SYSTEM DASDA1 (* System Configuration *)
  (* Standard: 61499-1 *)
  (* Version 0.4, 2009-03-05, JHC, Holobloc Inc., Deleted Application. *)
  (* Version 0.3, 2003-12-05, JHC, Rockwell Automation, Renamed from NEWSYSTEM. *)
  (* Version 0.2, 2002-11-05, JHC, Rockwell Automation, Fixed missing (empty) FBD in Application. *)
  (* Version 0.1, 2002-01-17, JHC, Rockwell Automation, Minor cleanup *)
  (* Version 0.0, 2000-05-27, JHC, Rockwell Automation *)
  DEVICE HMI_LAYER : FRAME_DEVICE(BOUNDS := [0,0,200,600])
    RESOURCE HMI_up : PANEL_RESOURCE(COLS := 1, ROWS := 10)
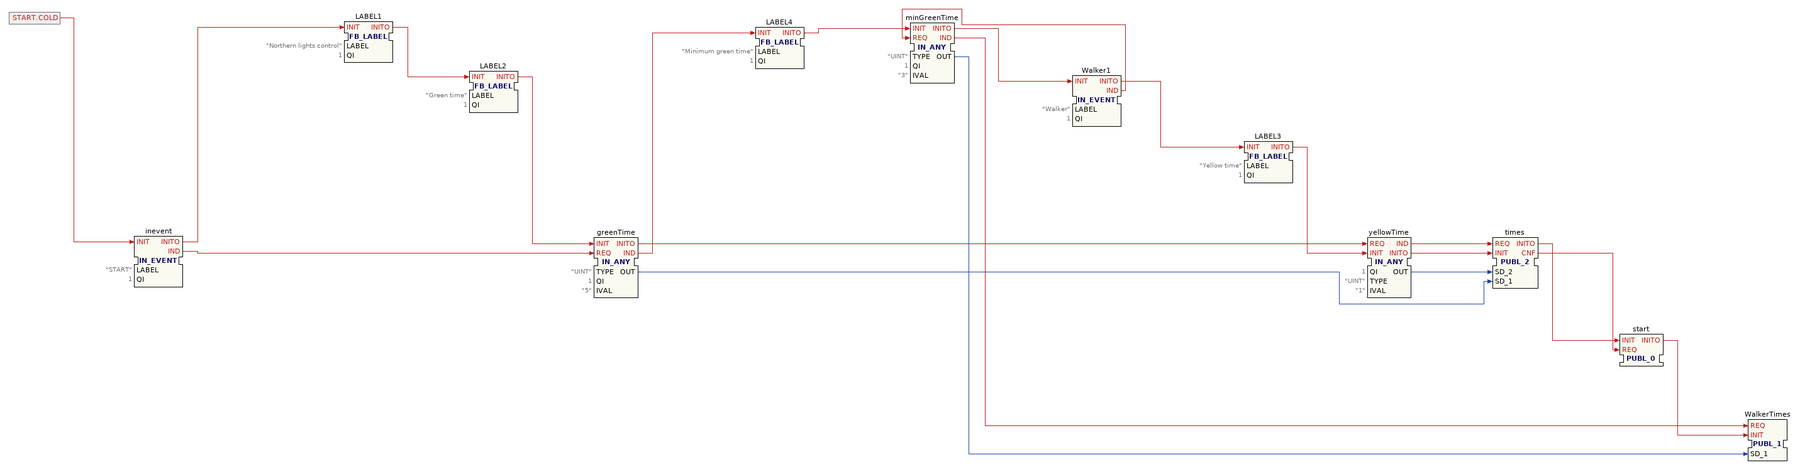
      FBS
        start : PUBL_0;
        greenTime : IN_ANY(TYPE := "UINT", QI := 1, IVAL := "5");
        yellowTime : IN_ANY(QI := 1, TYPE := "UINT", IVAL := "1");
        times : PUBL_2;
        LABEL1 : FB_LABEL(LABEL := "Northern lights control", QI := 1);
        LABEL2 : FB_LABEL(LABEL := "Green time", QI := 1);
        LABEL3 : FB_LABEL(LABEL := "Yellow time", QI := 1);
        minGreenTime : IN_ANY(TYPE := "UINT", QI := 1, IVAL := "3");
        LABEL4 : FB_LABEL(LABEL := "Minimum green time", QI := 1);
        Walker1 : IN_EVENT(LABEL := "Walker", QI := 1);
        WalkerTimes : PUBL_1;
        inevent : IN_EVENT(LABEL := "START", QI := 1);
      END_FBS
      EVENT_CONNECTIONS
        yellowTime.IND TO times.REQ;
        LABEL1.INITO TO LABEL2.INIT;
        LABEL2.INITO TO greenTime.INIT;
        greenTime.INITO TO LABEL4.INIT;
        LABEL4.INITO TO minGreenTime.INIT;
        greenTime.IND TO yellowTime.REQ;
        yellowTime.INITO TO times.INIT;
        times.INITO TO start.INIT;
        times.CNF TO start.REQ;
        minGreenTime.INITO TO Walker1.INIT;
        Walker1.INITO TO LABEL3.INIT;
        LABEL3.INITO TO yellowTime.INIT;
        Walker1.IND TO minGreenTime.REQ;
        minGreenTime.IND TO WalkerTimes.REQ;
        start.INITO TO WalkerTimes.INIT;
        START.COLD TO inevent.INIT;
        inevent.INITO TO LABEL1.INIT;
        inevent.IND TO greenTime.REQ;
      END_CONNECTIONS
      DATA_CONNECTIONS
        yellowTime.OUT TO times.SD_2;
        greenTime.OUT TO times.SD_1;
        minGreenTime.OUT TO WalkerTimes.SD_1;
      END_CONNECTIONS
    END_RESOURCE
    RESOURCE HMI_left : PANEL_RESOURCE(COLS := 1, ROWS := 10)
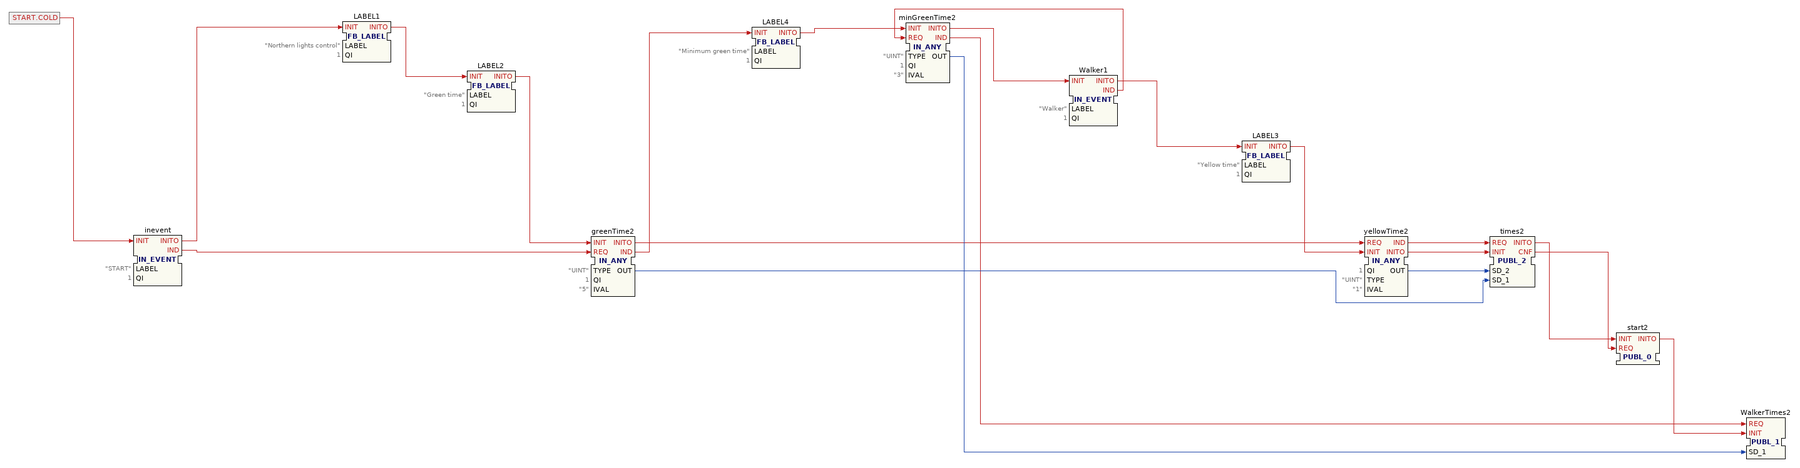
      FBS
        start2 : PUBL_0;
        greenTime2 : IN_ANY(TYPE := "UINT", QI := 1, IVAL := "5");
        yellowTime2 : IN_ANY(QI := 1, TYPE := "UINT", IVAL := "1");
        times2 : PUBL_2;
        LABEL1 : FB_LABEL(LABEL := "Northern lights control", QI := 1);
        LABEL2 : FB_LABEL(LABEL := "Green time", QI := 1);
        LABEL3 : FB_LABEL(LABEL := "Yellow time", QI := 1);
        minGreenTime2 : IN_ANY(TYPE := "UINT", QI := 1, IVAL := "3");
        LABEL4 : FB_LABEL(LABEL := "Minimum green time", QI := 1);
        Walker1 : IN_EVENT(LABEL := "Walker", QI := 1);
        WalkerTimes2 : PUBL_1;
        inevent : IN_EVENT(LABEL := "START", QI := 1);
      END_FBS
      EVENT_CONNECTIONS
        yellowTime2.IND TO times2.REQ;
        LABEL1.INITO TO LABEL2.INIT;
        LABEL2.INITO TO greenTime2.INIT;
        greenTime2.INITO TO LABEL4.INIT;
        LABEL4.INITO TO minGreenTime2.INIT;
        greenTime2.IND TO yellowTime2.REQ;
        yellowTime2.INITO TO times2.INIT;
        times2.INITO TO start2.INIT;
        times2.CNF TO start2.REQ;
        minGreenTime2.INITO TO Walker1.INIT;
        Walker1.INITO TO LABEL3.INIT;
        LABEL3.INITO TO yellowTime2.INIT;
        Walker1.IND TO minGreenTime2.REQ;
        minGreenTime2.IND TO WalkerTimes2.REQ;
        start2.INITO TO WalkerTimes2.INIT;
        START.COLD TO inevent.INIT;
        inevent.INITO TO LABEL1.INIT;
        inevent.IND TO greenTime2.REQ;
      END_CONNECTIONS
      DATA_CONNECTIONS
        yellowTime2.OUT TO times2.SD_2;
        greenTime2.OUT TO times2.SD_1;
        minGreenTime2.OUT TO WalkerTimes2.SD_1;
      END_CONNECTIONS
    END_RESOURCE
  END_DEVICE
  DEVICE MODEL_LAYER : FRAME_DEVICE
    RESOURCE LIGHTS_U : PANEL_RESOURCE
      FBS
        LightsControl : PUBL_3;
        start : SUBL_0;
        times : SUBL_2;
        LightsRT : PUBL_2;
        WalkerTimes : SUBL_1;
        LC1 : LIGHTS_CYCLE;
      END_FBS
      EVENT_CONNECTIONS
        START.COLD TO times.INIT;
        LightsControl.CNF TO LightsRT.REQ;
        start.INITO TO LightsControl.INIT;
        LightsControl.INITO TO LightsRT.INIT;
        times.INITO TO WalkerTimes.INIT;
        WalkerTimes.INITO TO start.INIT;
        start.IND TO LC1.START;
        WalkerTimes.IND TO LC1.WALKER;
        LC1.CNF TO LightsControl.REQ;
      END_CONNECTIONS
      DATA_CONNECTIONS
        WalkerTimes.RD_1 TO LC1.WALKERT;
        times.RD_1 TO LC1.GREENT;
        times.RD_2 TO LC1.YELLOWT;
        LC1.GREENOUT TO LightsControl.SD_1;
        LC1.YELLOWOUT TO LightsControl.SD_2;
        LC1.REDOUT TO LightsControl.SD_3;
        LC1.GREENRT TO LightsRT.SD_1;
        LC1.YELLOWRT TO LightsRT.SD_2;
      END_CONNECTIONS
    END_RESOURCE
    RESOURCE LIGHTS_L : PANEL_RESOURCE
      FBS
        LightsControl2 : PUBL_3;
        start2 : SUBL_0;
        times2 : SUBL_2;
        LightsRT2 : PUBL_2;
        WalkerTimes2 : SUBL_1;
        LC2 : LIGHTS_CYCLE;
      END_FBS
      EVENT_CONNECTIONS
        START.COLD TO times2.INIT;
        LightsControl2.CNF TO LightsRT2.REQ;
        start2.INITO TO LightsControl2.INIT;
        LightsControl2.INITO TO LightsRT2.INIT;
        times2.INITO TO WalkerTimes2.INIT;
        WalkerTimes2.INITO TO start2.INIT;
        start2.IND TO LC2.START;
        WalkerTimes2.IND TO LC2.WALKER;
        LC2.CNF TO LightsControl2.REQ;
      END_CONNECTIONS
      DATA_CONNECTIONS
        WalkerTimes2.RD_1 TO LC2.WALKERT;
        times2.RD_1 TO LC2.GREENT;
        times2.RD_2 TO LC2.YELLOWT;
        LC2.GREENOUT TO LightsControl2.SD_1;
        LC2.YELLOWOUT TO LightsControl2.SD_2;
        LC2.REDOUT TO LightsControl2.SD_3;
        LC2.GREENRT TO LightsRT2.SD_1;
        LC2.YELLOWRT TO LightsRT2.SD_2;
      END_CONNECTIONS
    END_RESOURCE
  END_DEVICE
  DEVICE VIEW_LAYER : FRAME_DEVICE(BOUNDS := [200,0,630,400], GRID := [1,1])
    RESOURCE view_res : PANEL_RESOURCE
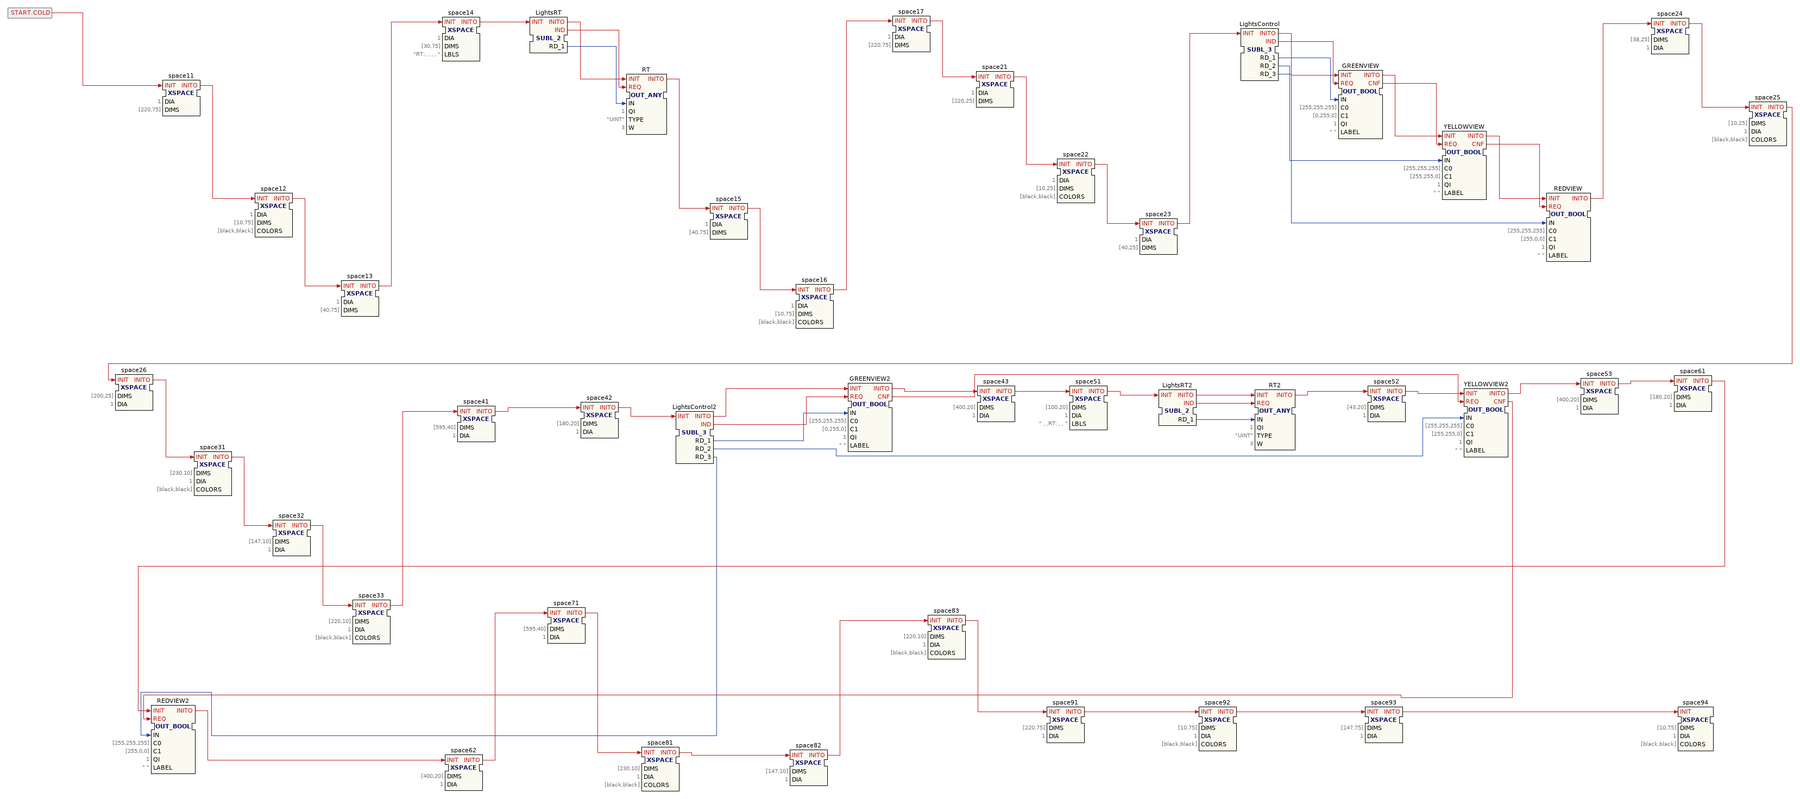
      FBS
        LightsControl : SUBL_3;
        GREENVIEW : OUT_BOOL(C0 := [255,255,255], C1 := [0,255,0], QI := 1, LABEL := " ");
        YELLOWVIEW : OUT_BOOL(C0 := [255,255,255], C1 := [255,255,0], QI := 1, LABEL := " ");
        REDVIEW : OUT_BOOL(C0 := [255,255,255], C1 := [255,0,0], QI := 1, LABEL := " ");
        space11 : XSPACE(DIA := 1, DIMS := [220,75]);
        space12 : XSPACE(DIA := 1, DIMS := [10,75], COLORS := [black,black]);
        space13 : XSPACE(DIA := 1, DIMS := [40,75]);
        space16 : XSPACE(DIA := 1, DIMS := [10,75], COLORS := [black,black]);
        space17 : XSPACE(DIA := 1, DIMS := [220,75]);
        space21 : XSPACE(DIA := 1, DIMS := [220,25]);
        space22 : XSPACE(DIA := 1, DIMS := [10,25], COLORS := [black,black]);
        space23 : XSPACE(DIA := 1, DIMS := [40,25]);
        space24 : XSPACE(DIMS := [38,25], DIA := 1);
        space25 : XSPACE(DIMS := [10,25], DIA := 1, COLORS := [black,black]);
        LightsRT : SUBL_2;
        space14 : XSPACE(DIA := 1, DIMS := [30,75], LBLS := "RT:, , , , ");
        RT : OUT_ANY(QI := 1, TYPE := "UINT", W := 3);
        space15 : XSPACE(DIA := 1, DIMS := [40,75]);
        space26 : XSPACE(DIMS := [200,25], DIA := 1);
        space31 : XSPACE(DIMS := [230,10], DIA := 1, COLORS := [black,black]);
        space32 : XSPACE(DIMS := [147,10], DIA := 1);
        space33 : XSPACE(DIMS := [220,10], DIA := 1, COLORS := [black,black]);
        space41 : XSPACE(DIMS := [595,40], DIA := 1);
        space42 : XSPACE(DIMS := [180,20], DIA := 1);
        LightsControl2 : SUBL_3;
        GREENVIEW2 : OUT_BOOL(C0 := [255,255,255], C1 := [0,255,0], QI := 1, LABEL := " ");
        space43 : XSPACE(DIMS := [400,20], DIA := 1);
        space51 : XSPACE(DIMS := [100,20], DIA := 1, LBLS := " , ,RT: , , ");
        LightsRT2 : SUBL_2;
        RT2 : OUT_ANY(QI := 1, TYPE := "UINT", W := 3);
        space52 : XSPACE(DIMS := [43,20], DIA := 1);
        YELLOWVIEW2 : OUT_BOOL(C0 := [255,255,255], C1 := [255,255,0], QI := 1, LABEL := " ");
        space53 : XSPACE(DIMS := [400,20], DIA := 1);
        space61 : XSPACE(DIMS := [180,20], DIA := 1);
        REDVIEW2 : OUT_BOOL(C0 := [255,255,255], C1 := [255,0,0], QI := 1, LABEL := " ");
        space62 : XSPACE(DIMS := [400,20], DIA := 1);
        space71 : XSPACE(DIMS := [595,40], DIA := 1);
        space81 : XSPACE(DIMS := [230,10], DIA := 1, COLORS := [black,black]);
        space82 : XSPACE(DIMS := [147,10], DIA := 1);
        space83 : XSPACE(DIMS := [220,10], DIA := 1, COLORS := [black,black]);
        space91 : XSPACE(DIMS := [220,75], DIA := 1);
        space92 : XSPACE(DIMS := [10,75], DIA := 1, COLORS := [black,black]);
        space93 : XSPACE(DIMS := [147,75], DIA := 1);
        space94 : XSPACE(DIMS := [10,75], DIA := 1, COLORS := [black,black]);
      END_FBS
      EVENT_CONNECTIONS
        LightsControl.INITO TO GREENVIEW.INIT;
        GREENVIEW.INITO TO YELLOWVIEW.INIT;
        YELLOWVIEW.INITO TO REDVIEW.INIT;
        LightsControl.IND TO GREENVIEW.REQ;
        GREENVIEW.CNF TO YELLOWVIEW.REQ;
        YELLOWVIEW.CNF TO REDVIEW.REQ;
        START.COLD TO space11.INIT;
        space11.INITO TO space12.INIT;
        space12.INITO TO space13.INIT;
        space16.INITO TO space17.INIT;
        space17.INITO TO space21.INIT;
        space21.INITO TO space22.INIT;
        space22.INITO TO space23.INIT;
        space23.INITO TO LightsControl.INIT;
        REDVIEW.INITO TO space24.INIT;
        space24.INITO TO space25.INIT;
        space13.INITO TO space14.INIT;
        space14.INITO TO LightsRT.INIT;
        LightsRT.INITO TO RT.INIT;
        LightsRT.IND TO RT.REQ;
        RT.INITO TO space15.INIT;
        space15.INITO TO space16.INIT;
        space25.INITO TO space26.INIT;
        space26.INITO TO space31.INIT;
        space31.INITO TO space32.INIT;
        space32.INITO TO space33.INIT;
        space33.INITO TO space41.INIT;
        space41.INITO TO space42.INIT;
        space42.INITO TO LightsControl2.INIT;
        LightsControl2.INITO TO GREENVIEW2.INIT;
        LightsControl2.IND TO GREENVIEW2.REQ;
        GREENVIEW2.INITO TO space43.INIT;
        space43.INITO TO space51.INIT;
        space51.INITO TO LightsRT2.INIT;
        LightsRT2.INITO TO RT2.INIT;
        LightsRT2.IND TO RT2.REQ;
        RT2.INITO TO space52.INIT;
        space52.INITO TO YELLOWVIEW2.INIT;
        YELLOWVIEW2.INITO TO space53.INIT;
        space53.INITO TO space61.INIT;
        space61.INITO TO REDVIEW2.INIT;
        REDVIEW2.INITO TO space62.INIT;
        space62.INITO TO space71.INIT;
        space71.INITO TO space81.INIT;
        space81.INITO TO space82.INIT;
        space82.INITO TO space83.INIT;
        space83.INITO TO space91.INIT;
        space91.INITO TO space92.INIT;
        space92.INITO TO space93.INIT;
        space93.INITO TO space94.INIT;
        GREENVIEW2.CNF TO YELLOWVIEW2.REQ;
        YELLOWVIEW2.CNF TO REDVIEW2.REQ;
      END_CONNECTIONS
      DATA_CONNECTIONS
        LightsControl.RD_1 TO GREENVIEW.IN;
        LightsControl.RD_2 TO YELLOWVIEW.IN;
        LightsControl.RD_3 TO REDVIEW.IN;
        LightsRT.RD_1 TO RT.IN;
        LightsControl2.RD_1 TO GREENVIEW2.IN;
        LightsControl2.RD_2 TO YELLOWVIEW2.IN;
        LightsControl2.RD_3 TO REDVIEW2.IN;
        LightsRT2.RD_1 TO RT2.IN;
      END_CONNECTIONS
    END_RESOURCE
  END_DEVICE
END_SYSTEM
